};
P[585]{
   GP1:
	UF : 1, UT : 1,		CONFIG : 'N U T, 0, 0, 0',
	X =  2337.679  mm,	Y =    42.631  mm,	Z =   847.798  mm,
	W =    36.871 deg,	P =    25.909 deg,	R =   -30.339 deg
   GP2:
	UF : 1, UT : 1,
	J1=    90.000 deg,	J2=   -90.000 deg
};
P[586]{
   GP1:
	UF : 1, UT : 1,		CONFIG : 'N U T, 0, 0, 0',
	X =  2406.124  mm,	Y =    41.236  mm,	Z =   848.781  mm,
	W =    37.791 deg,	P =    26.520 deg,	R =   -29.933 deg
   GP2:
	UF : 1, UT : 1,
	J1=    90.000 deg,	J2=   -90.000 deg
};
P[587]{
   GP1:
	UF : 1, UT : 1,		CONFIG : 'N U T, 0, 0, 0',
	X =  2410.910  mm,	Y =    45.622  mm,	Z =   847.064  mm,
	W =    14.866 deg,	P =    42.980 deg,	R =    21.274 deg
   GP2:
	UF : 1, UT : 1,
	J1=    90.000 deg,	J2=   -90.000 deg
};
P[588]{
   GP1:
	UF : 1, UT : 1,		CONFIG : 'N U T, 0, 0, 0',
	X =  2410.910  mm,	Y =    68.050  mm,	Z =   847.063  mm,
	W =    14.866 deg,	P =    42.980 deg,	R =    21.274 deg
   GP2:
	UF : 1, UT : 1,
	J1=    90.000 deg,	J2=   -90.000 deg
};
P[589]{
   GP1:
	UF : 1, UT : 1,		CONFIG : 'N U T, 0, 0, 0',
	X =  2465.746  mm,	Y =   547.387  mm,	Z =    91.178  mm,
	W =    16.836 deg,	P =   -31.148 deg,	R =   -30.329 deg
   GP2:
	UF : 1, UT : 1,
	J1=    80.000 deg,	J2=   -90.000 deg
};
P[590]{
   GP1:
	UF : 1, UT : 1,		CONFIG : 'N U T, 0, 0, 0',
	X =  2010.131  mm,	Y =   -94.796  mm,	Z =    -4.171  mm,
	W =    39.951 deg,	P =    24.695 deg,	R =    73.312 deg
   GP2:
	UF : 1, UT : 1,
	J1=    90.000 deg,	J2=  -100.000 deg
};
P[591]{
   GP1:
	UF : 1, UT : 1,		CONFIG : 'N U T, 0, 0, 0',
	X =  2008.984  mm,	Y =    22.770  mm,	Z =   -24.522  mm,
	W =    39.950 deg,	P =    24.717 deg,	R =    73.324 deg
   GP2:
	UF : 1, UT : 1,
	J1=    90.000 deg,	J2=  -100.000 deg
};
P[592]{
   GP1:
	UF : 1, UT : 1,		CONFIG : 'N U T, 0, 0, 0',
	X =  2263.191  mm,	Y =   -60.998  mm,	Z =     5.530  mm,
	W =    43.410 deg,	P =    13.252 deg,	R =    -7.762 deg
   GP2:
	UF : 1, UT : 1,
	J1=    90.000 deg,	J2=   -90.000 deg
};
P[593]{
   GP1:
	UF : 1, UT : 1,		CONFIG : 'N U T, 0, 0, 0',
	X =  2229.762  mm,	Y =   -61.641  mm,	Z =     5.530  mm,
	W =    43.410 deg,	P =    13.252 deg,	R =    -7.762 deg
   GP2:
	UF : 1, UT : 1,
	J1=    90.000 deg,	J2=   -90.000 deg
};
P[594]{
   GP1:
	UF : 1, UT : 1,		CONFIG : 'N U T, 0, 0, 0',
	X =  2140.673  mm,	Y =   -58.252  mm,	Z =    -4.687  mm,
	W =    43.401 deg,	P =    13.250 deg,	R =   -15.039 deg
   GP2:
	UF : 1, UT : 1,
	J1=    90.000 deg,	J2=   -90.000 deg
};
P[595]{
   GP1:
	UF : 1, UT : 1,		CONFIG : 'N U T, 0, 0, 0',
	X =  2202.385  mm,	Y =   -59.979  mm,	Z =    -2.526  mm,
	W =    43.410 deg,	P =    13.252 deg,	R =   -15.042 deg
   GP2:
	UF : 1, UT : 1,
	J1=    90.000 deg,	J2=   -90.000 deg
};
P[596]{
   GP1:
	UF : 1, UT : 1,		CONFIG : 'N U T, 0, 0, 0',
	X =  2214.325  mm,	Y =   -60.465  mm,	Z =    -2.403  mm,
	W =    43.410 deg,	P =    13.252 deg,	R =   -24.946 deg
   GP2:
	UF : 1, UT : 1,
	J1=    90.000 deg,	J2=   -90.000 deg
};
P[597]{
   GP1:
	UF : 1, UT : 1,		CONFIG : 'N U T, 0, 0, 0',
	X =  1993.391  mm,	Y =   -60.455  mm,	Z =   -13.196  mm,
	W =    43.411 deg,	P =    13.253 deg,	R =   -13.621 deg
   GP2:
	UF : 1, UT : 1,
	J1=    90.000 deg,	J2=   -90.000 deg
};
P[598]{
   GP1:
	UF : 1, UT : 1,		CONFIG : 'N U T, 0, 0, 0',
	X =  2091.686  mm,	Y =   -61.863  mm,	Z =   -12.523  mm,
	W =    43.411 deg,	P =    13.253 deg,	R =   -13.621 deg
   GP2:
	UF : 1, UT : 1,
	J1=    90.000 deg,	J2=   -90.000 deg
};
P[599]{
   GP1:
	UF : 1, UT : 1,		CONFIG : 'N U T, 0, 0, 0',
	X =  2578.421  mm,	Y =   578.735  mm,	Z =     1.160  mm,
	W =   -34.514 deg,	P =   -13.805 deg,	R =    35.075 deg
   GP2:
	UF : 1, UT : 1,
	J1=    80.000 deg,	J2=   -90.000 deg
};
P[600]{
   GP1:
	UF : 1, UT : 1,		CONFIG : 'N U T, 0, 0, 0',
	X =  2250.563  mm,	Y =   578.735  mm,	Z =   206.874  mm,
	W =   -34.514 deg,	P =   -13.805 deg,	R =    35.075 deg
   GP2:
	UF : 1, UT : 1,
	J1=    80.000 deg,	J2=   -90.000 deg
};
P[601]{
   GP1:
	UF : 1, UT : 1,		CONFIG : 'N U T, 0, 0, 0',
	X =  1581.308  mm,	Y =   447.592  mm,	Z =   359.920  mm,
	W =   -39.823 deg,	P =   -20.635 deg,	R =    36.563 deg
   GP2:
	UF : 1, UT : 1,
	J1=    80.000 deg,	J2=   -90.000 deg
};
P[602]{
   GP1:
	UF : 1, UT : 1,		CONFIG : 'N U T, 0, 0, 0',
	X =   966.134  mm,	Y =   141.704  mm,	Z =  1243.874  mm,
	W =   -10.927 deg,	P =      .883 deg,	R =    -9.877 deg
   GP2:
	UF : 1, UT : 1,
	J1=    80.000 deg,	J2=   -90.000 deg
};
P[603]{
   GP1:
	UF : 1, UT : 1,		CONFIG : 'N U T, 0, 0, 0',
	X =  1460.087  mm,	Y = -1490.374  mm,	Z =  1570.421  mm,
	W =    14.952 deg,	P =   -64.091 deg,	R =   -22.785 deg
   GP2:
	UF : 0, UT : 1,
	J1=   100.000 deg,	J2=   -90.000 deg
};
P[604]{
   GP1:
	UF : 1, UT : 1,		CONFIG : 'N U T, 0, 0, -1',
	X =  2509.757  mm,	Y = -1496.585  mm,	Z =  1047.977  mm,
	W =   -50.284 deg,	P =   -30.325 deg,	R =    67.097 deg
   GP2:
	UF : 0, UT : 1,
	J1=   100.000 deg,	J2=   -90.000 deg
};
P[605]{
   GP1:
	UF : 1, UT : 1,		CONFIG : 'N U T, 0, 0, 0',
	X =  2114.809  mm,	Y =   -65.234  mm,	Z =    -7.269  mm,
	W =    44.993 deg,	P =     6.743 deg,	R =   -31.685 deg
   GP2:
	UF : 1, UT : 1,
	J1=    90.000 deg,	J2=   -90.000 deg
};
P[606]{
   GP1:
	UF : 1, UT : 1,		CONFIG : 'N U T, 0, 0, 0',
	X =  2071.250  mm,	Y =  -111.352  mm,	Z =   -10.601  mm,
	W =   -38.374 deg,	P =    21.350 deg,	R =    99.173 deg
   GP2:
	UF : 1, UT : 1,
	J1=    90.000 deg,	J2=   -90.000 deg
};
P[607]{
   GP1:
	UF : 1, UT : 1,		CONFIG : 'N U T, 0, 0, 0',
	X =  2102.381  mm,	Y =   -81.362  mm,	Z =    -8.878  mm,
	W =   -38.373 deg,	P =    21.370 deg,	R =   110.629 deg
   GP2:
	UF : 1, UT : 1,
	J1=    90.000 deg,	J2=   -90.000 deg
};
P[608]{
   GP1:
	UF : 1, UT : 1,		CONFIG : 'N U T, 0, 0, 0',
	X =  2115.926  mm,	Y =   -68.888  mm,	Z =    -8.351  mm,
	W =   -38.378 deg,	P =    21.372 deg,	R =   123.344 deg
   GP2:
	UF : 1, UT : 1,
	J1=    90.000 deg,	J2=   -90.000 deg
};
P[609]{
   GP1:
	UF : 1, UT : 1,		CONFIG : 'N U T, 0, 0, 0',
	X =  2113.055  mm,	Y =  -234.031  mm,	Z =   836.605  mm,
	W =    -2.879 deg,	P =    40.084 deg,	R =   -96.451 deg
   GP2:
	UF : 1, UT : 1,
	J1=    90.000 deg,	J2=   -90.000 deg
};
P[610]{
   GP1:
	UF : 1, UT : 1,		CONFIG : 'N U T, 0, 0, 0',
	X =  2243.434  mm,	Y =  -233.025  mm,	Z =   836.634  mm,
	W =    -2.881 deg,	P =    40.072 deg,	R =   -96.452 deg
   GP2:
	UF : 1, UT : 1,
	J1=    90.000 deg,	J2=   -90.000 deg
};
P[611]{
   GP1:
	UF : 1, UT : 1,		CONFIG : 'N U T, 0, 0, 0',
	X =  2267.378  mm,	Y =  -226.582  mm,	Z =   836.634  mm,
	W =    -2.881 deg,	P =    40.072 deg,	R =   -66.779 deg
   GP2:
	UF : 1, UT : 1,
	J1=    90.000 deg,	J2=   -90.000 deg
};
P[612]{
   GP1:
	UF : 1, UT : 1,		CONFIG : 'N U T, 0, 0, 0',
	X =  2287.592  mm,	Y =  -213.439  mm,	Z =   836.634  mm,
	W =    -2.169 deg,	P =    44.406 deg,	R =   -56.318 deg
   GP2:
	UF : 1, UT : 1,
	J1=    90.000 deg,	J2=   -90.000 deg
};
P[613]{
   GP1:
	UF : 1, UT : 1,		CONFIG : 'N U T, 0, 0, 0',
	X =  2604.246  mm,	Y = -1559.689  mm,	Z =  1072.916  mm,
	W =   -42.880 deg,	P =   -14.276 deg,	R =     5.349 deg
   GP2:
	UF : 1, UT : 1,
	J1=   100.000 deg,	J2=   -90.000 deg
};
P[614]{
   GP1:
	UF : 1, UT : 1,		CONFIG : 'N U T, 0, 0, 0',
	X =  2404.490  mm,	Y = -1554.283  mm,	Z =  1178.815  mm,
	W =   -45.666 deg,	P =   -14.828 deg,	R =     8.688 deg
   GP2:
	UF : 1, UT : 1,
	J1=   100.000 deg,	J2=   -90.000 deg
};
P[615]{
   GP1:
	UF : 1, UT : 1,		CONFIG : 'N U T, 0, 0, 0',
	X =   310.715  mm,	Y =  -926.292  mm,	Z =  2102.112  mm,
	W =    13.518 deg,	P =   -46.200 deg,	R =   -44.908 deg
   GP2:
	UF : 1, UT : 1,
	J1=   180.000 deg,	J2=  -150.000 deg
};
P[616]{
   GP1:
	UF : 1, UT : 1,		CONFIG : 'N U T, 0, 0, 0',
	X =   411.688  mm,	Y = -1212.483  mm,	Z =  1529.953  mm,
	W =    32.650 deg,	P =   -32.880 deg,	R =   -50.053 deg
   GP2:
	UF : 1, UT : 1,
	J1=   180.000 deg,	J2=  -150.000 deg
};
P[617]{
   GP1:
	UF : 1, UT : 1,		CONFIG : 'N U T, 0, 0, 0',
	X =  1022.561  mm,	Y = -1112.994  mm,	Z =   854.309  mm,
	W =    32.649 deg,	P =   -32.880 deg,	R =   -22.647 deg
   GP2:
	UF : 1, UT : 1,
	J1=   180.000 deg,	J2=  -150.000 deg
};
P[618]{
   GP1:
	UF : 1, UT : 1,		CONFIG : 'N U T, 0, 0, 0',
	X =  2627.082  mm,	Y =    66.873  mm,	Z =   839.075  mm,
	W =    20.543 deg,	P =    38.277 deg,	R =   -21.061 deg
   GP2:
	UF : 1, UT : 1,
	J1=    90.000 deg,	J2=   -90.000 deg
};
P[619]{
   GP1:
	UF : 1, UT : 1,		CONFIG : 'N U T, 0, 0, 0',
	X =  2717.203  mm,	Y =   135.284  mm,	Z =   842.434  mm,
	W =    26.176 deg,	P =    38.126 deg,	R =   -54.891 deg
   GP2:
	UF : 1, UT : 1,
	J1=    90.000 deg,	J2=   -90.000 deg
};
P[620]{
   GP1:
	UF : 1, UT : 1,		CONFIG : 'N U T, 0, 0, 0',
	X =  1020.561  mm,	Y = -1102.994  mm,	Z =   866.309  mm,
	W =    32.649 deg,	P =   -32.880 deg,	R =   -22.647 deg
   GP2:
	UF : 1, UT : 1,
	J1=   180.000 deg,	J2=  -150.000 deg
};
P[621]{
   GP1:
	UF : 1, UT : 1,		CONFIG : 'N U T, 0, 0, 0',
	X =   743.145  mm,	Y =  -624.994  mm,	Z =   866.309  mm,
	W =   -10.474 deg,	P =   -44.020 deg,	R =    41.976 deg
   GP2:
	UF : 1, UT : 1,
	J1=   180.000 deg,	J2=  -150.000 deg
};
P[622]{
   GP1:
	UF : 1, UT : 1,		CONFIG : 'N U T, 0, 0, 0',
	X =  2132.094  mm,	Y =  -166.305  mm,	Z =   835.348  mm,
	W =      .273 deg,	P =    41.132 deg,	R =  -157.429 deg
   GP2:
	UF : 1, UT : 1,
	J1=    90.000 deg,	J2=   -90.000 deg
};
P[623]{
   GP1:
	UF : 1, UT : 1,		CONFIG : 'N U T, 0, 0, 0',
	X =  2121.423  mm,	Y =  -142.564  mm,	Z =   839.385  mm,
	W =      .273 deg,	P =    41.133 deg,	R =  -157.429 deg
   GP2:
	UF : 1, UT : 1,
	J1=    90.000 deg,	J2=   -90.000 deg
};
P[624]{
   GP1:
	UF : 1, UT : 1,		CONFIG : 'N U T, 0, 0, 0',
	X =   974.924  mm,	Y = -1071.847  mm,	Z =   858.131  mm,
	W =    40.735 deg,	P =   -21.063 deg,	R =   -37.349 deg
   GP2:
	UF : 1, UT : 1,
	J1=   180.000 deg,	J2=  -150.000 deg
};
P[625]{
   GP1:
	UF : 1, UT : 1,		CONFIG : 'N U T, 0, 0, 0',
	X =   535.748  mm,	Y =  -560.848  mm,	Z =   858.131  mm,
	W =     6.193 deg,	P =   -44.662 deg,	R =    21.224 deg
   GP2:
	UF : 1, UT : 1,
	J1=   180.000 deg,	J2=  -150.000 deg
};
P[626]{
   GP1:
	UF : 1, UT : 1,		CONFIG : 'N U T, 0, 0, 0',
	X =  2098.795  mm,	Y =  -128.635  mm,	Z =   838.528  mm,
	W =      .273 deg,	P =    41.131 deg,	R =   -73.876 deg
   GP2:
	UF : 1, UT : 1,
	J1=    90.000 deg,	J2=   -90.000 deg
};
P[627]{
   GP1:
	UF : 1, UT : 1,		CONFIG : 'N U T, 0, 0, 0',
	X =  2079.936  mm,	Y =  -151.778  mm,	Z =   834.671  mm,
	W =      .273 deg,	P =    41.131 deg,	R =    24.329 deg
   GP2:
	UF : 1, UT : 1,
	J1=    90.000 deg,	J2=   -90.000 deg
};
P[628]{
   GP1:
	UF : 1, UT : 1,		CONFIG : 'N U T, 0, 0, 0',
	X =   501.047  mm,	Y =  -783.398  mm,	Z =  1089.593  mm,
	W =    41.299 deg,	P =   -10.785 deg,	R =   -56.863 deg
   GP2:
	UF : 1, UT : 1,
	J1=   180.000 deg,	J2=  -150.000 deg
};
P[629]{
   GP1:
	UF : 1, UT : 1,		CONFIG : 'N U T, 0, 0, 0',
	X =  2093.049  mm,	Y =  -193.635  mm,	Z =   834.242  mm,
	W =      .273 deg,	P =    41.131 deg,	R =    24.329 deg
   GP2:
	UF : 1, UT : 1,
	J1=    90.000 deg,	J2=   -90.000 deg
};
P[630]{
   GP1:
	UF : 1, UT : 1,		CONFIG : 'N U T, 0, 0, 0',
	X =  2123.726  mm,	Y =  -207.135  mm,	Z =   835.200  mm,
	W =      .272 deg,	P =    41.130 deg,	R =   113.461 deg
   GP2:
	UF : 1, UT : 1,
	J1=    90.000 deg,	J2=   -90.000 deg
};
P[631]{
   GP1:
	UF : 1, UT : 1,		CONFIG : 'N U T, 0, 0, 0',
	X =  2137.679  mm,	Y =  1266.350  mm,	Z =   265.845  mm,
	W =    -1.526 deg,	P =    -1.652 deg,	R =     2.925 deg
   GP2:
	UF : 1, UT : 1,
	J1=    95.000 deg,	J2=    90.000 deg
};
P[632]{
   GP1:
	UF : 1, UT : 1,		CONFIG : 'N U T, 0, 0, 0',
	X =  2865.444  mm,	Y =  1350.388  mm,	Z =   109.119  mm,
	W =    -1.525 deg,	P =    -1.650 deg,	R =     2.923 deg
   GP2:
	UF : 1, UT : 1,
	J1=    95.000 deg,	J2=    90.000 deg
};
P[633]{
   GP1:
	UF : 1, UT : 1,		CONFIG : 'N U T, 0, 0, 1',
	X =  2135.638  mm,	Y =  -181.420  mm,	Z =   836.815  mm,
	W =      .272 deg,	P =    41.129 deg,	R =  -155.380 deg
   GP2:
	UF : 1, UT : 1,
	J1=    90.000 deg,	J2=   -90.000 deg
};
P[634]{
   GP1:
	UF : 1, UT : 1,		CONFIG : 'N U T, 0, 0, 0',
	X =  2860.268  mm,	Y =  1355.846  mm,	Z =    75.220  mm,
	W =    -1.278 deg,	P =    -1.674 deg,	R =     2.900 deg
   GP2:
	UF : 1, UT : 1,
	J1=    94.999 deg,	J2=    90.000 deg
};
P[635]{
   GP1:
	UF : 1, UT : 1,		CONFIG : 'N U T, 0, 0, 0',
	X =  2378.751  mm,	Y =  1298.143  mm,	Z =   191.223  mm,
	W =    -1.364 deg,	P =    -1.667 deg,	R =     2.909 deg
   GP2:
	UF : 1, UT : 1,
	J1=    94.999 deg,	J2=    90.000 deg
};
P[636]{
   GP1:
	UF : 1, UT : 1,		CONFIG : 'N U T, 0, 0, 0',
	X =  1491.977  mm,	Y =  1529.258  mm,	Z =  1071.362  mm,
	W =    42.682 deg,	P =    16.600 deg,	R =   -42.377 deg
   GP2:
	UF : 1, UT : 1,
	J1=    95.000 deg,	J2=    90.000 deg
};
P[637]{
   GP1:
	UF : 1, UT : 1,		CONFIG : 'N U T, 0, 0, 1',
	X =  2131.366  mm,	Y =  -167.649  mm,	Z =   836.816  mm,
	W =      .273 deg,	P =    41.129 deg,	R =  -155.380 deg
   GP2:
	UF : 1, UT : 1,
	J1=    90.000 deg,	J2=   -90.000 deg
};
P[638]{
   GP1:
	UF : 1, UT : 1,		CONFIG : 'N U T, 0, 0, 0',
	X =  1962.457  mm,	Y =   -45.639  mm,	Z =    58.921  mm,
	W =   -44.047 deg,	P =    11.474 deg,	R =    22.771 deg
   GP2:
	UF : 1, UT : 1,
	J1=    90.000 deg,	J2=   -90.000 deg
};
P[639]{
   GP1:
	UF : 1, UT : 1,		CONFIG : 'N U T, 0, 0, 0',
	X =  1938.711  mm,	Y =   -47.041  mm,	Z =    57.874  mm,
	W =   -44.064 deg,	P =    11.483 deg,	R =     9.318 deg
   GP2:
	UF : 1, UT : 1,
	J1=    90.000 deg,	J2=   -90.000 deg
};
P[640]{
   GP1:
	UF : 1, UT : 1,		CONFIG : 'N U T, 0, 0, 0',
	X =  1695.757  mm,	Y =   -46.889  mm,	Z =    59.031  mm,
	W =   -44.062 deg,	P =    11.485 deg,	R =     9.319 deg
   GP2:
	UF : 1, UT : 1,
	J1=    90.000 deg,	J2=   -90.000 deg
};
P[641]{
   GP1:
	UF : 1, UT : 1,		CONFIG : 'N U T, 0, 0, 0',
	X =  1672.272  mm,	Y =   -45.995  mm,	Z =    59.374  mm,
	W =   -42.428 deg,	P =     8.383 deg,	R =   -27.316 deg
   GP2:
	UF : 1, UT : 1,
	J1=    90.000 deg,	J2=   -90.000 deg
};
P[642]{
   GP1:
	UF : 1, UT : 1,		CONFIG : 'N U T, 0, 0, 0',
	X =  2227.243  mm,	Y =   -48.667  mm,	Z =     3.919  mm,
	W =   -43.618 deg,	P =    12.240 deg,	R =    12.516 deg
   GP2:
	UF : 1, UT : 1,
	J1=    90.000 deg,	J2=   -90.000 deg
};
P[643]{
   GP1:
	UF : 1, UT : 1,		CONFIG : 'N U T, 0, 0, 0',
	X =   918.608  mm,	Y =    -7.834  mm,	Z =  2170.036  mm,
	W =     -.013 deg,	P =   -45.002 deg,	R =     -.002 deg
   GP2:
	UF : 1, UT : 1,
	J1=     0.000 deg,	J2=   -40.000 deg
};
P[644]{
   GP1:
	UF : 1, UT : 1,		CONFIG : 'N U T, 0, 0, 0',
	X =  1048.055  mm,	Y = -1040.484  mm,	Z =  1492.639  mm,
	W =   -30.893 deg,	P =    38.446 deg,	R =    21.262 deg
   GP2:
	UF : 1, UT : 1,
	J1=   180.000 deg,	J2=   -90.000 deg
};
P[645]{
   GP1:
	UF : 1, UT : 1,		CONFIG : 'N U T, 0, 0, 0',
	X =  1872.811  mm,	Y = -1301.247  mm,	Z =  1254.086  mm,
	W =   -41.810 deg,	P =   -20.894 deg,	R =   -21.724 deg
   GP2:
	UF : 0, UT : 1,
	J1=   180.000 deg,	J2=   -90.000 deg
};
P[646]{
   GP1:
	UF : 1, UT : 1,		CONFIG : 'N U T, 0, 0, 0',
	X =  1938.810  mm,	Y = -1402.247  mm,	Z =  1047.086  mm,
	W =   -42.701 deg,	P =    18.644 deg,	R =    19.122 deg
   GP2:
	UF : 0, UT : 1,
	J1=   180.000 deg,	J2=   -90.000 deg
};
P[647]{
   GP1:
	UF : 1, UT : 1,		CONFIG : 'N U T, 0, 0, 0',
	X =  2268.430  mm,	Y =   -49.062  mm,	Z =     3.148  mm,
	W =   -43.638 deg,	P =    12.235 deg,	R =    12.536 deg
   GP2:
	UF : 1, UT : 1,
	J1=    90.000 deg,	J2=   -90.000 deg
};
P[648]{
   GP1:
	UF : 1, UT : 1,		CONFIG : 'N U T, 0, 0, 0',
	X =  2144.289  mm,	Y =   -44.663  mm,	Z =    -3.347  mm,
	W =   -43.586 deg,	P =    12.233 deg,	R =    12.506 deg
   GP2:
	UF : 1, UT : 1,
	J1=    90.000 deg,	J2=   -90.000 deg
};
P[649]{
   GP1:
	UF : 1, UT : 1,		CONFIG : 'N U T, 0, 0, 0',
	X =  2206.737  mm,	Y =   -44.800  mm,	Z =    -4.310  mm,
	W =   -43.648 deg,	P =    12.245 deg,	R =    12.536 deg
   GP2:
	UF : 1, UT : 1,
	J1=    90.000 deg,	J2=   -90.000 deg
};
P[650]{
   GP1:
	UF : 1, UT : 1,		CONFIG : 'N U T, 0, 0, 0',
	X =  2215.198  mm,	Y =   -41.335  mm,	Z =    -1.874  mm,
	W =   -43.835 deg,	P =    12.332 deg,	R =    22.820 deg
   GP2:
	UF : 1, UT : 1,
	J1=    90.000 deg,	J2=   -90.000 deg
};
P[651]{
   GP1:
	UF : 1, UT : 1,		CONFIG : 'N U T, 0, 0, 0',
	X =  2048.302  mm,	Y = -1378.190  mm,	Z =  1060.194  mm,
	W =   -44.862 deg,	P =     3.961 deg,	R =   -20.537 deg
   GP2:
	UF : 0, UT : 1,
	J1=   180.000 deg,	J2=   -90.000 deg
};
P[652]{
   GP1:
	UF : 1, UT : 1,		CONFIG : 'N U T, 0, 0, 0',
	X =  1872.811  mm,	Y = -1301.247  mm,	Z =  1254.086  mm,
	W =   -41.810 deg,	P =   -20.894 deg,	R =   -21.724 deg
   GP2:
	UF : 0, UT : 1,
	J1=   180.000 deg,	J2=   -90.000 deg
};
P[653]{
   GP1:
	UF : 1, UT : 1,		CONFIG : 'N U T, 0, 0, 0',
	X =  1690.020  mm,	Y = -1301.247  mm,	Z =  1305.059  mm,
	W =   -41.810 deg,	P =   -20.894 deg,	R =   -21.725 deg
   GP2:
	UF : 0, UT : 1,
	J1=   180.000 deg,	J2=   -90.000 deg
};
P[654]{
   GP1:
	UF : 1, UT : 1,		CONFIG : 'N U T, 0, 0, 0',
	X =  1677.457  mm,	Y = -1378.259  mm,	Z =  1040.446  mm,
	W =   -45.888 deg,	P =   -20.593 deg,	R =    49.871 deg
   GP2:
	UF : 1, UT : 1,
	J1=   180.000 deg,	J2=  -125.000 deg
};
P[655]{
   GP1:
	UF : 1, UT : 1,		CONFIG : 'N U T, 0, 0, 0',
	X =  1566.667  mm,	Y =  1053.178  mm,	Z =  1535.870  mm,
	W =    48.261 deg,	P =    -8.333 deg,	R =     1.925 deg
   GP2:
	UF : 1, UT : 1,
	J1=   180.000 deg,	J2=    90.000 deg
};
P[656]{
   GP1:
	UF : 1, UT : 1,		CONFIG : 'N U T, 0, 0, 0',
	X =  1858.811  mm,	Y =  1224.223  mm,	Z =  1340.087  mm,
	W =    44.958 deg,	P =    -2.212 deg,	R =     2.229 deg
   GP2:
	UF : 0, UT : 1,
	J1=   180.000 deg,	J2=    90.000 deg
};
P[657]{
   GP1:
	UF : 1, UT : 1,		CONFIG : 'N U T, 0, 0, 0',
	X =  1935.691  mm,	Y =  1358.717  mm,	Z =  1058.831  mm,
	W =    41.277 deg,	P =    19.800 deg,	R =   -21.086 deg
   GP2:
	UF : 0, UT : 1,
	J1=   180.000 deg,	J2=    90.000 deg
};
P[658]{
   GP1:
	UF : 1, UT : 1,		CONFIG : 'N U T, 0, 0, 0',
	X =  2117.652  mm,	Y =   -48.970  mm,	Z =   -12.273  mm,
	W =   -43.851 deg,	P =     1.342 deg,	R =     1.316 deg
   GP2:
	UF : 1, UT : 1,
	J1=    90.000 deg,	J2=   -90.000 deg
};
P[659]{
   GP1:
	UF : 1, UT : 1,		CONFIG : 'N U T, 0, 0, 0',
	X =  2046.175  mm,	Y =   -49.955  mm,	Z =   -12.492  mm,
	W =   -43.835 deg,	P =     1.333 deg,	R =     1.297 deg
   GP2:
	UF : 1, UT : 1,
	J1=    89.999 deg,	J2=   -90.000 deg
};
P[660]{
   GP1:
	UF : 1, UT : 1,		CONFIG : 'N U T, 0, 0, 0',
	X =  2016.609  mm,	Y =   -47.854  mm,	Z =   -12.356  mm,
	W =   -43.890 deg,	P =     1.338 deg,	R =   -18.633 deg
   GP2:
	UF : 1, UT : 1,
	J1=    90.000 deg,	J2=   -90.000 deg
};
P[661]{
   GP1:
	UF : 1, UT : 1,		CONFIG : 'N U T, 0, 0, 0',
	X =  1655.760  mm,	Y =   145.124  mm,	Z =   -12.456  mm,
	W =     1.625 deg,	P =    45.218 deg,	R =  -176.807 deg
   GP2:
	UF : 1, UT : 1,
	J1=    90.000 deg,	J2=   -90.000 deg
};
P[662]{
   GP1:
	UF : 1, UT : 1,		CONFIG : 'N U T, 0, 0, 0',
	X =  2002.299  mm,	Y =  1434.488  mm,	Z =  1057.303  mm,
	W =    44.305 deg,	P =     8.850 deg,	R =     3.803 deg
   GP2:
	UF : 1, UT : 1,
	J1=   180.000 deg,	J2=    90.000 deg
};
P[663]{
   GP1:
	UF : 1, UT : 1,		CONFIG : 'N U T, 0, 0, 0',
	X =  1858.811  mm,	Y =  1224.223  mm,	Z =  1340.087  mm,
	W =    44.958 deg,	P =    -2.212 deg,	R =     2.229 deg
   GP2:
	UF : 0, UT : 1,
	J1=   180.000 deg,	J2=    90.000 deg
};
P[664]{
   GP1:
	UF : 1, UT : 1,		CONFIG : 'N U T, 0, 0, 0',
	X =  1606.614  mm,	Y = -1413.568  mm,	Z =  1053.901  mm,
	W =   -44.560 deg,	P =   -18.266 deg,	R =    45.822 deg
   GP2:
	UF : 1, UT : 1,
	J1=   180.000 deg,	J2=  -125.000 deg
};
P[665]{
   GP1:
	UF : 1, UT : 1,		CONFIG : 'N U T, 0, 0, 0',
	X =  1539.706  mm,	Y = -1470.455  mm,	Z =  1071.063  mm,
	W =   -42.856 deg,	P =   -15.293 deg,	R =    39.131 deg
   GP2:
	UF : 1, UT : 1,
	J1=   180.000 deg,	J2=  -125.000 deg
};
P[666]{
   GP1:
	UF : 1, UT : 1,		CONFIG : 'N U T, 0, 0, 0',
	X =  1128.196  mm,	Y = -1374.012  mm,	Z =  1522.225  mm,
	W =   -32.586 deg,	P =   -12.067 deg,	R =    17.529 deg
   GP2:
	UF : 1, UT : 1,
	J1=   180.000 deg,	J2=  -125.000 deg
};
P[667]{
   GP1:
	UF : 1, UT : 1,		CONFIG : 'N U T, 0, 0, 0',
	X =  1322.021  mm,	Y =   -61.275  mm,	Z =  2053.615  mm,
	W =     5.182 deg,	P =   -69.521 deg,	R =     3.554 deg
   GP2:
	UF : 1, UT : 1,
	J1=   180.000 deg,	J2=  -125.000 deg
};
P[668]{
   GP1:
	UF : 1, UT : 1,		CONFIG : 'N U T, 0, 0, 0',
	X =   160.262  mm,	Y = -1423.433  mm,	Z =   468.198  mm,
	W =   -49.202 deg,	P =    -2.428 deg,	R =     4.065 deg
   GP2:
	UF : 1, UT : 1,
	J1=    80.000 deg,	J2=    90.000 deg
};
P[669]{
   GP1:
	UF : 1, UT : 1,		CONFIG : 'N U T, 0, 0, 0',
	X =  1898.966  mm,	Y = -1114.290  mm,	Z =   250.136  mm,
	W =   -43.355 deg,	P =    13.455 deg,	R =    94.693 deg
   GP2:
	UF : 1, UT : 1,
	J1=    90.000 deg,	J2=   -90.000 deg
};
P[670]{
   GP1:
	UF : 1, UT : 1,		CONFIG : 'N U T, 0, 0, 0',
	X =  1553.976  mm,	Y =  -228.945  mm,	Z =  1213.332  mm,
	W =     5.098 deg,	P =    43.299 deg,	R =   155.065 deg
   GP2:
	UF : 1, UT : 1,
	J1=    90.000 deg,	J2=   -90.000 deg
};
P[671]{
   GP1:
	UF : 1, UT : 1,		CONFIG : 'N U T, 0, 0, 0',
	X =  1293.632  mm,	Y =   272.064  mm,	Z =   747.059  mm,
	W =   -29.792 deg,	P =   -24.153 deg,	R =    10.342 deg
   GP2:
	UF : 1, UT : 1,
	J1=    80.000 deg,	J2=   -90.000 deg
};
P[672]{
   GP1:
	UF : 1, UT : 1,		CONFIG : 'N U T, 0, 0, 0',
	X =  1934.301  mm,	Y = -1340.280  mm,	Z =  1676.218  mm,
	W =   -39.185 deg,	P =   -21.096 deg,	R =     2.457 deg
   GP2:
	UF : 1, UT : 1,
	J1=   100.000 deg,	J2=   -90.000 deg
};
P[673]{
   GP1:
	UF : 1, UT : 1,		CONFIG : 'N U T, 0, 0, 0',
	X =  1863.859  mm,	Y =  -353.796  mm,	Z =   377.216  mm,
	W =     -.805 deg,	P =    13.426 deg,	R =    -8.574 deg
   GP2:
	UF : 1, UT : 1,
	J1=    90.000 deg,	J2=  -134.989 deg
};
P[674]{
   GP1:
	UF : 1, UT : 1,		CONFIG : 'N U T, 0, 0, 0',
	X =  1657.899  mm,	Y =   -24.482  mm,	Z =   -13.743  mm,
	W =    35.889 deg,	P =    31.029 deg,	R =  -138.190 deg
   GP2:
	UF : 1, UT : 1,
	J1=    90.000 deg,	J2=   -90.000 deg
};
P[675]{
   GP1:
	UF : 1, UT : 1,		CONFIG : 'N U T, 0, 0, 0',
	X =  2067.448  mm,	Y =   -40.115  mm,	Z =    22.547  mm,
	W =    34.294 deg,	P =    -8.375 deg,	R =   -88.174 deg
   GP2:
	UF : 1, UT : 1,
	J1=    80.000 deg,	J2=   -90.000 deg
};
P[676]{
   GP1:
	UF : 1, UT : 1,		CONFIG : 'N U T, 0, 0, 0',
	X =  2071.895  mm,	Y =    -9.046  mm,	Z =    21.479  mm,
	W =    34.239 deg,	P =    -8.411 deg,	R =   -88.218 deg
   GP2:
	UF : 1, UT : 1,
	J1=    80.000 deg,	J2=   -90.000 deg
};
P[677]{
   GP1:
	UF : 1, UT : 1,		CONFIG : 'N U T, 0, 0, 0',
	X =  2076.271  mm,	Y =     4.342  mm,	Z =    21.635  mm,
	W =    30.086 deg,	P =   -21.642 deg,	R =   -96.023 deg
   GP2:
	UF : 1, UT : 1,
	J1=    80.000 deg,	J2=   -90.000 deg
};
P[678]{
   GP1:
	UF : 1, UT : 1,		CONFIG : 'N U T, 0, 0, 0',
	X =  2086.260  mm,	Y =    16.914  mm,	Z =    21.636  mm,
	W =    23.411 deg,	P =   -33.701 deg,	R =  -102.541 deg
   GP2:
	UF : 1, UT : 1,
	J1=    80.000 deg,	J2=   -90.000 deg
};
P[679]{
   GP1:
	UF : 1, UT : 1,		CONFIG : 'N U T, 0, 0, 0',
	X =  2099.624  mm,	Y =    22.343  mm,	Z =    16.408  mm,
	W =    23.412 deg,	P =   -33.704 deg,	R =  -102.541 deg
   GP2:
	UF : 1, UT : 1,
	J1=    80.000 deg,	J2=   -90.000 deg
};
P[680]{
   GP1:
	UF : 1, UT : 1,		CONFIG : 'N U T, 0, 0, 0',
	X =  2111.220  mm,	Y =    30.146  mm,	Z =    16.113  mm,
	W =    23.413 deg,	P =   -33.667 deg,	R =   -79.616 deg
   GP2:
	UF : 1, UT : 1,
	J1=    80.000 deg,	J2=   -90.000 deg
};
P[681]{
   GP1:
	UF : 1, UT : 1,		CONFIG : 'N U T, 0, 0, 0',
	X =  2117.747  mm,	Y =    34.877  mm,	Z =    15.620  mm,
	W =    21.330 deg,	P =   -32.904 deg,	R =   -59.466 deg
   GP2:
	UF : 1, UT : 1,
	J1=    80.000 deg,	J2=   -90.000 deg
};
P[682]{
   GP1:
	UF : 1, UT : 1,		CONFIG : 'N U T, 0, 0, 0',
	X =  2637.097  mm,	Y =   276.051  mm,	Z =   -70.874  mm,
	W =    26.007 deg,	P =   -23.136 deg,	R =   -26.934 deg
   GP2:
	UF : 1, UT : 1,
	J1=    80.000 deg,	J2=   -90.000 deg
};
P[683]{
   GP1:
	UF : 1, UT : 1,		CONFIG : 'N U T, 0, 0, 0',
	X =  2631.473  mm,	Y =   295.376  mm,	Z =   -71.289  mm,
	W =    23.061 deg,	P =   -24.098 deg,	R =   -27.768 deg
   GP2:
	UF : 1, UT : 1,
	J1=    80.000 deg,	J2=   -90.000 deg
};
P[684]{
   GP1:
	UF : 1, UT : 1,		CONFIG : 'N U T, 0, 0, 0',
	X =  2630.839  mm,	Y =   309.534  mm,	Z =   -72.681  mm,
	W =    13.725 deg,	P =   -26.025 deg,	R =   -27.412 deg
   GP2:
	UF : 1, UT : 1,
	J1=    80.000 deg,	J2=   -90.000 deg
};
P[685]{
   GP1:
	UF : 1, UT : 1,		CONFIG : 'F U T, 0, 0, 0',
	X =  2688.926  mm,	Y =   145.792  mm,	Z =   479.238  mm,
	W =    11.537 deg,	P =   -44.440 deg,	R =    16.356 deg
   GP2:
	UF : 1, UT : 1,
	J1=    90.000 deg,	J2=     0.000 deg
};
P[686]{
   GP1:
	UF : 1, UT : 1,		CONFIG : 'N U T, 0, 0, 0',
	X =  2629.380  mm,	Y =   555.199  mm,	Z =   -71.771  mm,
	W =    16.234 deg,	P =   -30.277 deg,	R =   -30.022 deg
   GP2:
	UF : 1, UT : 1,
	J1=    80.000 deg,	J2=   -90.000 deg
};
P[687]{
   GP1:
	UF : 1, UT : 1,		CONFIG : 'N U T, 0, 0, 0',
	X =  2774.631  mm,	Y =   -50.226  mm,	Z =  -585.366  mm,
	W =    -7.964 deg,	P =    29.527 deg,	R =   -15.865 deg
   GP2:
	UF : 1, UT : 1,
	J1=    90.000 deg,	J2=     -.000 deg
};
P[688]{
   GP1:
	UF : 1, UT : 1,		CONFIG : 'N U T, 0, 0, 0',
	X =  1299.331  mm,	Y = -1307.282  mm,	Z =    76.272  mm,
	W =     -.716 deg,	P =    46.671 deg,	R =  -161.579 deg
   GP2:
	UF : 1, UT : 1,
	J1=     -.000 deg,	J2=   -40.000 deg
};
P[690]{
   GP1:
	UF : 1, UT : 1,		CONFIG : 'N U T, 0, 0, 0',
	X =  2025.246  mm,	Y =   179.636  mm,	Z =    77.704  mm,
	W =    44.528 deg,	P =     7.306 deg,	R =  -107.368 deg
   GP2:
	UF : 1, UT : 1,
	J1=    90.000 deg,	J2=    90.000 deg
};
P[691]{
   GP1:
	UF : 1, UT : 1,		CONFIG : 'N U T, 0, 0, 0',
	X =  1631.701  mm,	Y =   -36.025  mm,	Z =    10.513  mm,
	W =   -35.869 deg,	P =    29.234 deg,	R =   139.446 deg
   GP2:
	UF : 1, UT : 1,
	J1=    90.000 deg,	J2=    90.000 deg
};
P[692]{
   GP1:
	UF : 1, UT : 1,		CONFIG : 'N U T, 0, 0, 0',
	X =  2352.388  mm,	Y =    33.975  mm,	Z =    37.420  mm,
	W =    44.702 deg,	P =     5.823 deg,	R =    -5.853 deg
   GP2:
	UF : 1, UT : 1,
	J1=    90.000 deg,	J2=    90.000 deg
};
P[698]{
   GP1:
	UF : 1, UT : 1,		CONFIG : 'N U T, 0, 0, 0',
	X =  2556.356  mm,	Y =   671.307  mm,	Z =   -63.224  mm,
	W =    14.773 deg,	P =   -27.994 deg,	R =   -29.313 deg
   GP2:
	UF : 1, UT : 1,
	J1=    80.000 deg,	J2=   -90.000 deg
};
P[699]{
   GP1:
	UF : 1, UT : 1,		CONFIG : 'N U T, 0, 0, 0',
	X =  2527.768  mm,	Y =    82.975  mm,	Z =    35.040  mm,
	W =   -19.934 deg,	P =   -29.387 deg,	R =   -57.880 deg
   GP2:
	UF : 1, UT : 1,
	J1=    90.000 deg,	J2=   100.000 deg
};
P[700]{
   GP1:
	UF : 1, UT : 1,		CONFIG : 'N U T, 0, 0, 0',
	X =  2555.963  mm,	Y =   661.878  mm,	Z =   -63.273  mm,
	W =    14.820 deg,	P =   -28.053 deg,	R =   -29.338 deg
   GP2:
	UF : 1, UT : 1,
	J1=    80.000 deg,	J2=   -90.000 deg
};
P[701]{
   GP1:
	UF : 1, UT : 1,		CONFIG : 'N U T, 0, 0, 0',
	X =  2563.772  mm,	Y =   648.879  mm,	Z =   -60.031  mm,
	W =    37.349 deg,	P =    -1.493 deg,	R =   -59.573 deg
   GP2:
	UF : 1, UT : 1,
	J1=    79.999 deg,	J2=   -90.000 deg
};
P[702]{
   GP1:
	UF : 1, UT : 1,		CONFIG : 'N U T, 0, 0, 0',
	X =  2069.947  mm,	Y =   -19.018  mm,	Z =    71.892  mm,
	W =   -33.592 deg,	P =   -20.528 deg,	R =   113.872 deg
   GP2:
	UF : 1, UT : 1,
	J1=    80.000 deg,	J2=    90.000 deg
};
P[703]{
   GP1:
	UF : 1, UT : 1,		CONFIG : 'N U T, 0, 0, 0',
	X =  2581.702  mm,	Y =   645.887  mm,	Z =   -65.892  mm,
	W =    40.898 deg,	P =    15.309 deg,	R =   -28.288 deg
   GP2:
	UF : 1, UT : 1,
	J1=    79.999 deg,	J2=   -90.000 deg
};
P[704]{
   GP1:
	UF : 1, UT : 1,		CONFIG : 'N U T, 0, 0, 0',
	X =  2301.493  mm,	Y =  -174.041  mm,	Z =    77.114  mm,
	W =   -18.811 deg,	P =   -35.778 deg,	R =    80.101 deg
   GP2:
	UF : 1, UT : 1,
	J1=    80.000 deg,	J2=    90.000 deg
};
P[705]{
   GP1:
	UF : 1, UT : 1,		CONFIG : 'N U T, 0, 0, 0',
	X =  2391.169  mm,	Y =  -255.392  mm,	Z =    38.246  mm,
	W =   -31.684 deg,	P =   -29.665 deg,	R =   116.915 deg
   GP2:
	UF : 1, UT : 1,
	J1=    80.000 deg,	J2=    90.000 deg
};
P[706]{
   GP1:
	UF : 1, UT : 1,		CONFIG : 'N U T, 0, 0, 0',
	X =  2365.453  mm,	Y =  -173.250  mm,	Z =    -3.469  mm,
	W =   -24.610 deg,	P =   -35.578 deg,	R =   136.285 deg
   GP2:
	UF : 1, UT : 1,
	J1=    80.000 deg,	J2=    90.000 deg
};
P[707]{
   GP1:
	UF : 1, UT : 1,		CONFIG : 'N U T, 0, 0, 0',
	X =  2599.532  mm,	Y =   647.084  mm,	Z =   -71.487  mm,
	W =    36.219 deg,	P =    25.994 deg,	R =   -28.148 deg
   GP2:
	UF : 1, UT : 1,
	J1=    80.000 deg,	J2=   -90.000 deg
};
P[708]{
   GP1:
	UF : 1, UT : 1,		CONFIG : 'N U T, 0, 0, 0',
	X =  2639.652  mm,	Y =   617.545  mm,	Z =   -73.525  mm,
	W =    28.739 deg,	P =   -19.543 deg,	R =   -26.170 deg
   GP2:
	UF : 1, UT : 1,
	J1=    80.000 deg,	J2=   -90.000 deg
};
P[709]{
   GP1:
	UF : 1, UT : 1,		CONFIG : 'N U T, 0, 0, 0',
	X =  2633.078  mm,	Y =   565.134  mm,	Z =   -73.033  mm,
	W =   -30.056 deg,	P =   -21.487 deg,	R =    14.835 deg
   GP2:
	UF : 1, UT : 1,
	J1=    80.000 deg,	J2=   -90.000 deg
};
P[710]{
   GP1:
	UF : 1, UT : 1,		CONFIG : 'N U T, 0, 0, 0',
	X =  2627.231  mm,	Y =   559.955  mm,	Z =   -68.972  mm,
	W =   -30.241 deg,	P =   -22.146 deg,	R =    24.484 deg
   GP2:
	UF : 1, UT : 1,
	J1=    80.000 deg,	J2=   -90.000 deg
};
P[711]{
   GP1:
	UF : 1, UT : 1,		CONFIG : 'N U T, 1, 0, 0',
	X =  2626.492  mm,	Y =   555.669  mm,	Z =   -68.972  mm,
	W =   -30.241 deg,	P =   -22.146 deg,	R =    34.932 deg
   GP2:
	UF : 1, UT : 1,
	J1=    80.000 deg,	J2=   -90.000 deg
};
P[712]{
   GP1:
	UF : 1, UT : 1,		CONFIG : 'N U T, 0, 0, 0',
	X =  2226.536  mm,	Y =  -221.028  mm,	Z =   279.124  mm,
	W =    32.202 deg,	P =   -34.003 deg,	R =    80.899 deg
   GP2:
	UF : 1, UT : 1,
	J1=    90.000 deg,	J2=  -100.000 deg
};
P[713]{
   GP1:
	UF : 1, UT : 1,		CONFIG : 'N U T, 0, 0, 0',
	X =  2604.414  mm,	Y =   146.949  mm,	Z =   202.251  mm,
	W =    57.531 deg,	P =    -1.632 deg,	R =    14.147 deg
   GP2:
	UF : 1, UT : 1,
	J1=    90.000 deg,	J2=  -100.000 deg
};
P[714]{
   GP1:
	UF : 1, UT : 1,		CONFIG : 'N U T, 0, 0, 0',
	X =  2604.414  mm,	Y =   -97.338  mm,	Z =   134.395  mm,
	W =    11.998 deg,	P =   -34.016 deg,	R =    74.095 deg
   GP2:
	UF : 1, UT : 1,
	J1=    90.000 deg,	J2=  -100.000 deg
};
P[715]{
   GP1:
	UF : 1, UT : 1,		CONFIG : 'N U T, 0, 0, 0',
	X =  2786.086  mm,	Y = -1479.912  mm,	Z =   941.700  mm,
	W =   -37.794 deg,	P =   -31.379 deg,	R =    42.844 deg
   GP2:
	UF : 1, UT : 1,
	J1=   100.000 deg,	J2=   -90.000 deg
};
P[716]{
   GP1:
	UF : 1, UT : 1,		CONFIG : 'N U T, 0, 0, 0',
	X =  2786.986  mm,	Y = -1505.928  mm,	Z =   939.959  mm,
	W =   -37.771 deg,	P =   -31.405 deg,	R =    42.828 deg
   GP2:
	UF : 1, UT : 1,
	J1=   100.000 deg,	J2=   -90.000 deg
};
P[717]{
   GP1:
	UF : 1, UT : 1,		CONFIG : 'N U T, 0, 0, 0',
	X =  2774.678  mm,	Y = -1541.827  mm,	Z =   940.534  mm,
	W =   -42.873 deg,	P =   -22.986 deg,	R =    43.313 deg
   GP2:
	UF : 1, UT : 1,
	J1=   100.000 deg,	J2=   -90.000 deg
};
P[718]{
   GP1:
	UF : 1, UT : 1,		CONFIG : 'N U T, 0, 0, 0',
	X =  2764.543  mm,	Y = -1552.501  mm,	Z =   937.834  mm,
	W =   -45.718 deg,	P =   -14.892 deg,	R =    35.274 deg
   GP2:
	UF : 1, UT : 1,
	J1=   100.000 deg,	J2=   -90.000 deg
};
P[719]{
   GP1:
	UF : 1, UT : 1,		CONFIG : 'N U T, 0, 0, 0',
	X =  2726.183  mm,	Y = -1572.833  mm,	Z =   931.213  mm,
	W =   -45.718 deg,	P =   -14.891 deg,	R =    30.406 deg
   GP2:
	UF : 1, UT : 1,
	J1=   100.000 deg,	J2=   -90.000 deg
};
P[720]{
   GP1:
	UF : 1, UT : 1,		CONFIG : 'N U T, 0, 0, 0',
	X =  2715.419  mm,	Y = -1577.423  mm,	Z =   928.201  mm,
	W =   -45.718 deg,	P =   -14.891 deg,	R =    18.309 deg
   GP2:
	UF : 1, UT : 1,
	J1=   100.000 deg,	J2=   -90.000 deg
};
P[721]{
   GP1:
	UF : 1, UT : 1,		CONFIG : 'N U T, 0, 0, 0',
	X =  2708.762  mm,	Y = -1578.705  mm,	Z =   926.876  mm,
	W =   -45.671 deg,	P =   -14.925 deg,	R =     6.059 deg
   GP2:
	UF : 1, UT : 1,
	J1=   100.000 deg,	J2=   -90.000 deg
};
P[722]{
   GP1:
	UF : 1, UT : 1,		CONFIG : 'N U T, 0, 0, 1',
	X =  2112.580  mm,	Y =  -162.135  mm,	Z =   871.673  mm,
	W =      .273 deg,	P =    41.129 deg,	R =  -155.380 deg
   GP2:
	UF : 1, UT : 1,
	J1=    90.000 deg,	J2=   -90.000 deg
};
P[723]{
   GP1:
	UF : 1, UT : 1,		CONFIG : 'N U T, 0, 0, 0',
	X =  1934.190  mm,	Y =     8.768  mm,	Z =   115.651  mm,
	W =   -44.064 deg,	P =    11.483 deg,	R =    19.176 deg
   GP2:
	UF : 1, UT : 1,
	J1=    90.000 deg,	J2=   -90.000 deg
};
P[724]{
   GP1:
	UF : 1, UT : 1,		CONFIG : 'N U T, 0, 0, 0',
	X =  2674.922  mm,	Y = -1580.021  mm,	Z =   920.473  mm,
	W =   -43.507 deg,	P =   -15.103 deg,	R =     5.510 deg
   GP2:
	UF : 1, UT : 1,
	J1=   100.000 deg,	J2=   -90.000 deg
};
P[725]{
   GP1:
	UF : 1, UT : 1,		CONFIG : 'N U T, 0, 0, 0',
	X =  1059.676  mm,	Y = -1060.441  mm,	Z =   780.990  mm,
	W =    33.685 deg,	P =   -33.155 deg,	R =   -22.872 deg
   GP2:
	UF : 1, UT : 1,
	J1=   180.000 deg,	J2=  -150.000 deg
};
P[726]{
   GP1:
	UF : 1, UT : 1,		CONFIG : 'N U T, 0, 0, 0',
	X =  1100.173  mm,	Y = -1128.611  mm,	Z =   779.932  mm,
	W =    33.801 deg,	P =   -33.260 deg,	R =   -22.966 deg
   GP2:
	UF : 1, UT : 1,
	J1=   180.000 deg,	J2=  -150.000 deg
};
P[727]{
   GP1:
	UF : 1, UT : 1,		CONFIG : 'N U T, 0, 0, 0',
	X =   775.571  mm,	Y =  -578.980  mm,	Z =   775.648  mm,
	W =    -9.238 deg,	P =   -44.139 deg,	R =    41.976 deg
   GP2:
	UF : 1, UT : 1,
	J1=   180.000 deg,	J2=  -150.000 deg
};
P[728]{
   GP1:
	UF : 1, UT : 1,		CONFIG : 'N U T, 0, 0, 0',
	X =  1032.684  mm,	Y = -1029.380  mm,	Z =   776.764  mm,
	W =    -9.289 deg,	P =   -44.218 deg,	R =    42.018 deg
   GP2:
	UF : 1, UT : 1,
	J1=   180.000 deg,	J2=  -150.000 deg
};
P[729]{
   GP1:
	UF : 1, UT : 1,		CONFIG : 'N U T, 0, 0, 0',
	X =   716.770  mm,	Y =  -475.623  mm,	Z =   775.298  mm,
	W =     6.193 deg,	P =   -44.662 deg,	R =    21.224 deg
   GP2:
	UF : 1, UT : 1,
	J1=   180.000 deg,	J2=  -150.000 deg
};
P[730]{
   GP1:
	UF : 1, UT : 1,		CONFIG : 'N U T, 0, 0, 0',
	X =  2066.428  mm,	Y =    38.562  mm,	Z =    83.681  mm,
	W =    21.323 deg,	P =   -32.915 deg,	R =   -59.432 deg
   GP2:
	UF : 1, UT : 1,
	J1=    80.000 deg,	J2=   -90.000 deg
};
P[731]{
   GP1:
	UF : 1, UT : 1,		CONFIG : 'N U T, 0, 0, 0',
	X =  2170.000  mm,	Y =    97.491  mm,	Z =    83.679  mm,
	W =    21.322 deg,	P =   -32.914 deg,	R =  -104.338 deg
   GP2:
	UF : 1, UT : 1,
	J1=    80.000 deg,	J2=   -90.000 deg
};
P[732]{
   GP1:
	UF : 1, UT : 1,		CONFIG : 'N U T, 0, 0, 0',
	X =  2151.501  mm,	Y =    54.276  mm,	Z =    23.680  mm,
	W =    12.359 deg,	P =   -39.979 deg,	R =  -118.608 deg
   GP2:
	UF : 1, UT : 1,
	J1=    80.000 deg,	J2=   -90.000 deg
};
P[733]{
   GP1:
	UF : 1, UT : 1,		CONFIG : 'N U T, 0, 0, 0',
	X =   757.404  mm,	Y =  -544.801  mm,	Z =   775.425  mm,
	W =     6.193 deg,	P =   -44.662 deg,	R =    21.224 deg
   GP2:
	UF : 1, UT : 1,
	J1=   180.000 deg,	J2=  -150.000 deg
};
P[734]{
   GP1:
	UF : 1, UT : 1,		CONFIG : 'N U T, 0, 0, 0',
	X =  1897.493  mm,	Y = -1471.823  mm,	Z =  1034.427  mm,
	W =   -41.048 deg,	P =    21.456 deg,	R =    22.832 deg
   GP2:
	UF : 1, UT : 1,
	J1=   180.000 deg,	J2=   -90.000 deg
};
P[735]{
   GP1:
	UF : 1, UT : 1,		CONFIG : 'N U T, 0, 0, 0',
	X =  1926.995  mm,	Y = -1472.868  mm,	Z =  1037.670  mm,
	W =   -43.499 deg,	P =    14.501 deg,	R =    14.844 deg
   GP2:
	UF : 1, UT : 1,
	J1=   180.000 deg,	J2=   -90.000 deg
};
P[736]{
   GP1:
	UF : 1, UT : 1,		CONFIG : 'N U T, 0, 0, 0',
	X =  1961.292  mm,	Y = -1474.240  mm,	Z =  1036.908  mm,
	W =   -43.543 deg,	P =    14.555 deg,	R =    14.822 deg
   GP2:
	UF : 1, UT : 1,
	J1=   180.000 deg,	J2=   -90.000 deg
};
P[737]{
   GP1:
	UF : 1, UT : 1,		CONFIG : 'N U T, 0, 0, 0',
	X =  1981.198  mm,	Y = -1482.302  mm,	Z =  1036.170  mm,
	W =   -43.849 deg,	P =    14.842 deg,	R =    -4.649 deg
   GP2:
	UF : 1, UT : 1,
	J1=   180.000 deg,	J2=   -90.000 deg
};
P[738]{
   GP1:
	UF : 1, UT : 1,		CONFIG : 'N U T, 0, 0, 0',
	X =  1997.161  mm,	Y = -1496.181  mm,	Z =  1035.858  mm,
	W =   -43.543 deg,	P =    14.555 deg,	R =   -28.270 deg
   GP2:
	UF : 1, UT : 1,
	J1=   180.000 deg,	J2=   -90.000 deg
};
P[739]{
   GP1:
	UF : 1, UT : 1,		CONFIG : 'N U T, 0, 0, 0',
	X =  1898.587  mm,	Y =  1470.493  mm,	Z =  1038.822  mm,
	W =    41.338 deg,	P =    19.894 deg,	R =   -17.217 deg
   GP2:
	UF : 1, UT : 1,
	J1=   180.000 deg,	J2=    90.000 deg
};
P[740]{
   GP1:
	UF : 1, UT : 1,		CONFIG : 'N U T, 0, 0, 0',
	X =  1927.314  mm,	Y =  1470.795  mm,	Z =  1041.672  mm,
	W =    41.283 deg,	P =    19.814 deg,	R =   -17.227 deg
   GP2:
	UF : 1, UT : 1,
	J1=   180.000 deg,	J2=    90.000 deg
};
P[741]{
   GP1:
	UF : 1, UT : 1,		CONFIG : 'N U T, 0, 0, 0',
	X =  1965.969  mm,	Y =  1477.380  mm,	Z =  1035.803  mm,
	W =    41.278 deg,	P =    19.810 deg,	R =   -17.222 deg
   GP2:
	UF : 1, UT : 1,
	J1=   180.000 deg,	J2=    90.000 deg
};
P[742]{
   GP1:
	UF : 1, UT : 1,		CONFIG : 'F U T, 0, 0, 0',
	X =   813.665  mm,	Y =   984.387  mm,	Z =  1106.553  mm,
	W =    50.730 deg,	P =      .639 deg,	R =   -51.736 deg
   GP2:
	UF : 1, UT : 1,
	J1=   180.000 deg,	J2=   150.000 deg
};
P[743]{
   GP1:
	UF : 1, UT : 1,		CONFIG : 'F U T, 0, 0, 0',
	X =  1073.308  mm,	Y =  1002.601  mm,	Z =  1061.552  mm,
	W =    50.730 deg,	P =      .639 deg,	R =   -51.736 deg
   GP2:
	UF : 1, UT : 1,
	J1=   180.000 deg,	J2=   150.000 deg
};
P[744]{
   GP1:
	UF : 1, UT : 1,		CONFIG : 'N U T, 0, 0, 0',
	X =  1986.252  mm,	Y =  1485.948  mm,	Z =  1036.367  mm,
	W =    41.276 deg,	P =    19.802 deg,	R =     6.735 deg
   GP2:
	UF : 1, UT : 1,
	J1=   180.000 deg,	J2=    90.000 deg
};
P[745]{
   GP1:
	UF : 1, UT : 1,		CONFIG : 'N U T, 0, 0, 0',
	X =  1991.631  mm,	Y =  1485.776  mm,	Z =  1039.525  mm,
	W =    41.277 deg,	P =    19.801 deg,	R =    21.629 deg
   GP2:
	UF : 1, UT : 1,
	J1=   180.000 deg,	J2=    90.000 deg
};
P[746]{
   GP1:
	UF : 1, UT : 1,		CONFIG : 'N U T, 0, 0, 0',
	X =  1641.393  mm,	Y = -1413.503  mm,	Z =  1035.805  mm,
	W =   -42.856 deg,	P =   -15.294 deg,	R =    39.130 deg
   GP2:
	UF : 1, UT : 1,
	J1=   180.000 deg,	J2=  -125.000 deg
};
P[747]{
   GP1:
	UF : 1, UT : 1,		CONFIG : 'N U T, 0, 0, 0',
	X =  1644.977  mm,	Y = -1406.796  mm,	Z =  1036.157  mm,
	W =   -42.573 deg,	P =   -16.796 deg,	R =    40.474 deg
   GP2:
	UF : 1, UT : 1,
	J1=   180.000 deg,	J2=  -125.000 deg
};
P[748]{
   GP1:
	UF : 1, UT : 1,		CONFIG : 'F U T, 0, 0, 0',
	X =  1126.179  mm,	Y =   980.555  mm,	Z =  1056.327  mm,
	W =    50.535 deg,	P =   -23.426 deg,	R =   -25.981 deg
   GP2:
	UF : 1, UT : 1,
	J1=   180.000 deg,	J2=   150.000 deg
};
P[749]{
   GP1:
	UF : 1, UT : 1,		CONFIG : 'F U T, 0, 0, 0',
	X =   861.179  mm,	Y =   980.555  mm,	Z =  1056.327  mm,
	W =    50.535 deg,	P =   -23.426 deg,	R =   -25.981 deg
   GP2:
	UF : 1, UT : 1,
	J1=   180.000 deg,	J2=   150.000 deg
};
P[750]{
   GP1:
	UF : 1, UT : 1,		CONFIG : 'F U T, 0, 0, 0',
	X =   761.179  mm,	Y =  1040.555  mm,	Z =  1247.135  mm,
	W =    50.535 deg,	P =   -23.426 deg,	R =   -25.981 deg
   GP2:
	UF : 1, UT : 1,
	J1=   180.000 deg,	J2=   150.000 deg
};
P[751]{
   GP1:
	UF : 1, UT : 1,		CONFIG : 'N U T, 0, 0, 0',
	X =  1659.432  mm,	Y = -1394.615  mm,	Z =  1037.456  mm,
	W =   -42.573 deg,	P =   -16.796 deg,	R =    43.536 deg
   GP2:
	UF : 1, UT : 1,
	J1=   180.000 deg,	J2=  -125.000 deg
};
P[752]{
   GP1:
	UF : 1, UT : 1,		CONFIG : 'N U T, 0, 0, 0',
	X =  1683.235  mm,	Y = -1387.627  mm,	Z =  1038.136  mm,
	W =   -44.235 deg,	P =   -18.485 deg,	R =    48.309 deg
   GP2:
	UF : 1, UT : 1,
	J1=   180.000 deg,	J2=  -125.000 deg
};
P[753]{
   GP1:
	UF : 1, UT : 1,		CONFIG : 'F U T, 0, 0, 0',
	X =  1102.375  mm,	Y =  1006.778  mm,	Z =  1032.261  mm,
	W =    50.724 deg,	P =      .658 deg,	R =   -51.733 deg
   GP2:
	UF : 1, UT : 1,
	J1=   180.000 deg,	J2=   150.000 deg
};
P[754]{
   GP1:
	UF : 1, UT : 1,		CONFIG : 'F U T, 0, 0, 0',
	X =  1113.834  mm,	Y =   999.761  mm,	Z =  1032.940  mm,
	W =    50.730 deg,	P =      .639 deg,	R =   -51.736 deg
   GP2:
	UF : 1, UT : 1,
	J1=   180.000 deg,	J2=   150.000 deg
};
P[755]{
   GP1:
	UF : 1, UT : 1,		CONFIG : 'F U T, 0, 0, 0',
	X =  1127.114  mm,	Y =   997.098  mm,	Z =  1032.585  mm,
	W =    50.728 deg,	P =      .638 deg,	R =   -36.952 deg
   GP2:
	UF : 1, UT : 1,
	J1=   180.000 deg,	J2=   150.000 deg
};
P[756]{
   GP1:
	UF : 1, UT : 1,		CONFIG : 'N U B, 0, 0, 0',
	X =   356.008  mm,	Y =    -2.081  mm,	Z =  2424.081  mm,
	W =      .008 deg,	P =   -40.007 deg,	R =     -.004 deg
   GP2:
	UF : 1, UT : 1,
	J1=    45.000 deg,	J2=     0.000 deg
};
P[757]{
   GP1:
	UF : 1, UT : 1,		CONFIG : 'N U T, 0, 0, 0',
	X =   988.747  mm,	Y =  -208.560  mm,	Z =  2175.643  mm,
	W =     4.196 deg,	P =   -34.982 deg,	R =   -12.442 deg
   GP2:
	UF : 1, UT : 1,
	J1=   135.000 deg,	J2=     0.000 deg
};
P[758]{
   GP1:
	UF : 1, UT : 1,		CONFIG : 'F U T, 0, 0, 0',
	X =  1139.649  mm,	Y =   996.948  mm,	Z =  1033.938  mm,
	W =    48.461 deg,	P =   -17.355 deg,	R =   -20.268 deg
   GP2:
	UF : 1, UT : 1,
	J1=   180.000 deg,	J2=   150.000 deg
};
P[759]{
   GP1:
	UF : 1, UT : 1,		CONFIG : 'N U T, 0, 0, 0',
	X =  1921.096  mm,	Y =   -30.244  mm,	Z =   155.039  mm,
	W =     -.111 deg,	P =    22.917 deg,	R =     -.285 deg
   GP2:
	UF : 1, UT : 1,
	J1=    45.206 deg,	J2=   180.000 deg
};
P[760]{
   GP1:
	UF : 1, UT : 1,		CONFIG : 'N U B, 0, 0, 0',
	X =   356.032  mm,	Y =    -2.146  mm,	Z =  2424.049  mm,
	W =      .001 deg,	P =   -40.002 deg,	R =     -.005 deg
   GP2:
	UF : 1, UT : 1,
	J1=     0.000 deg,	J2=   180.000 deg
};
P[761]{
   GP1:
	UF : 1, UT : 1,		CONFIG : 'N U T, 0, 0, 0',
	X =  1435.319  mm,	Y =   360.965  mm,	Z =   608.631  mm,
	W =     3.160 deg,	P =   -22.165 deg,	R =   -20.317 deg
   GP2:
	UF : 1, UT : 1,
	J1=    90.000 deg,	J2=   135.000 deg
};
P[762]{
   GP1:
	UF : 1, UT : 1,		CONFIG : 'N U B, 0, 0, 0',
	X =   356.032  mm,	Y =    -2.146  mm,	Z =  2424.049  mm,
	W =      .001 deg,	P =   -40.002 deg,	R =     -.005 deg
   GP2:
	UF : 1, UT : 1,
	J1=    95.000 deg,	J2=    90.000 deg
};
P[763]{
   GP1:
	UF : 1, UT : 1,		CONFIG : 'N U T, 0, 0, 0',
	X =   950.520  mm,	Y =   205.285  mm,	Z =  1027.227  mm,
	W =    53.651 deg,	P =   -10.142 deg,	R =   -83.497 deg
   GP2:
	UF : 1, UT : 1,
	J1=   -90.000 deg,	J2=   -90.000 deg
};
P[764]{
   GP1:
	UF : 1, UT : 1,		CONFIG : 'N U T, 0, 0, 0',
	X =   918.607  mm,	Y =    -7.726  mm,	Z =  2170.023  mm,
	W =     -.002 deg,	P =   -45.001 deg,	R =     -.002 deg
   GP2:
	UF : 1, UT : 1,
	J1=   -90.000 deg,	J2=    90.000 deg
};
P[766]{
   GP1:
	UF : 1, UT : 1,		CONFIG : 'N U T, 0, 0, 0',
	X =  1192.014  mm,	Y =   363.761  mm,	Z =   366.390  mm,
	W =   -29.115 deg,	P =     8.226 deg,	R =     2.246 deg
   GP2:
	UF : 1, UT : 1,
	J1=    90.000 deg,	J2=   100.000 deg
};
P[769]{
   GP1:
	UF : 1, UT : 1,		CONFIG : 'N U B, 0, 0, 0',
	X =   355.995  mm,	Y =    -2.096  mm,	Z =  2424.051  mm,
	W =     -.002 deg,	P =   -40.003 deg,	R =      .002 deg
   GP2:
	UF : 1, UT : 1,
	J1=   100.000 deg,	J2=   -90.000 deg
};
P[771]{
   GP1:
	UF : 1, UT : 1,		CONFIG : 'N U T, 0, 0, 0',
	X =   373.078  mm,	Y =  -901.222  mm,	Z =  1248.293  mm,
	W =    40.112 deg,	P =    11.399 deg,	R =   -86.822 deg
   GP2:
	UF : 1, UT : 1,
	J1=   180.000 deg,	J2=  -150.000 deg
};
P[773]{
   GP1:
	UF : 1, UT : 1,		CONFIG : 'N U T, 0, 0, 0',
	X =  1672.878  mm,	Y =   916.398  mm,	Z =  1594.940  mm,
	W =    39.846 deg,	P =    -9.760 deg,	R =     1.478 deg
   GP2:
	UF : 1, UT : 1,
	J1=   180.000 deg,	J2=    90.000 deg
};
P[774]{
   GP1:
	UF : 1, UT : 1,		CONFIG : 'N U B, 0, 0, 0',
	X =   356.032  mm,	Y =    -2.147  mm,	Z =  2424.050  mm,
	W =      .001 deg,	P =   -40.002 deg,	R =     -.005 deg
   GP2:
	UF : 1, UT : 1,
	J1=   180.000 deg,	J2=   150.000 deg
};
P[777]{
   GP1:
	UF : 1, UT : 1,		CONFIG : 'N U T, 0, 0, 0',
	X =  1147.490  mm,	Y =   177.260  mm,	Z =   168.328  mm,
	W =    32.004 deg,	P =   -33.504 deg,	R =  -110.246 deg
   GP2:
	UF : 1, UT : 1,
	J1=    90.000 deg,	J2=    90.000 deg
};
P[783]{
   GP1:
	UF : 1, UT : 1,		CONFIG : 'F U T, 0, 0, 0',
	X =   419.331  mm,	Y =  1026.789  mm,	Z =  1609.020  mm,
	W =    71.318 deg,	P =     7.769 deg,	R =   -20.454 deg
   GP2:
	UF : 1, UT : 1,
	J1=   180.000 deg,	J2=   150.000 deg
};
/END
